(* IEC 61131-3 sources: json/test/Deserializer, 7 files *)

(* ---- Test_GetValues_Arrays.st ---- *)
USING Simatic.Ax.Conversion;
USING AxUnit.Assert;
USING System.Strings;
using Simatic.Ax.Json;

NAMESPACE Deserializer
NAMESPACE GetValues

{TestFixture}
CLASS Test_Deserializer_GetValues_Arrays
    VAR protected
        deserializer : Deserializer;

        buffer : ARRAY[0..999] OF CHAR;
        key: STRING;
        value: STRING;
    END_VAR

    {Test}
    Method Public Test_FindValue_in_JSON_SimpleArray
        VAR
            JSON_Entry: STRING := '{ "arraykey": [123, 456]}';

            len:DINT;
            keyFound: BOOL;
        END_VAR

        len:= Strings.ToArray(str := JSON_Entry, arr := buffer);
        deserializer.SetBuffer(REF(buffer)); //TODO: ausbauen und ersetzen durch buffer in methode

        key := 'arraykey';
        keyFound := deserializer.GetValue( REF(key), value);
        Equal('[123, 456]', value);
    END_Method

    {Test}
    Method Public Test_FindValue_in_JSON_ComplexArray
        VAR
            JSON_Entry: STRING := '{ "key1": 1234,"arraykey": [123, 456], "key2": 456}';

            len:DINT;
            keyFound: BOOL;
        END_VAR

        len:= Strings.ToArray(str := JSON_Entry, arr := buffer);
        deserializer.SetBuffer(REF(buffer)); //TODO: ausbauen und ersetzen durch buffer in methode

        key := 'arraykey';
        keyFound := deserializer.GetValue( REF(key), value);
        Equal('[123, 456]', value);
    END_Method

    {Test}
    Method Public Test_FindValue_in_JSON_NestedArray
        VAR
            JSON_Entry: STRING := '{ "key1": 1234,"arraykey": [{"nestedkey1": 1234, "nestedkey2": 456}, {"nestedkey3": 1234, "nestedkey4": 456}], "key2": 456}';

            len:DINT;
            keyFound: BOOL;
        END_VAR

        len:= Strings.ToArray(str := JSON_Entry, arr := buffer);
        deserializer.SetBuffer(REF(buffer)); //TODO: ausbauen und ersetzen durch buffer in methode

        key := 'arraykey';
        keyFound := deserializer.GetValue( REF(key), value);
        Equal('[{"nestedkey1": 1234, "nestedkey2": 456}, {"nestedkey3": 1234, "nestedkey4": 456}]', value);
    END_Method

END_CLASS

END_NAMESPACE
END_NAMESPACE

(* ---- Test_GetValues_NestedElements.st ---- *)
USING Simatic.Ax.Conversion;
USING AxUnit.Assert;
USING System.Strings;
using Simatic.Ax.Json;

NAMESPACE Deserializer
NAMESPACE GetValues

{TestFixture}
CLASS Test_Deserializer_GetValues_NestedElements
    VAR protected
        deserializer : Deserializer;

        buffer : ARRAY[0..999] OF CHAR;
        key: STRING;
        value: STRING;
    END_VAR

    {Test}
    Method Public Test_FindValue_in_JSON_NestedArray
        VAR
            JSON_Entry: STRING := '{ "key1": 1234,"arraykey": [{"nestedkey1": 1234, "nestedkey2": 456}, {"nestedkey3": 1234, "nestedkey4": 456}], "key2": 456}';

            len:DINT;
            keyFound: BOOL;
        END_VAR

        len:= Strings.ToArray(str := JSON_Entry, arr := buffer);
        deserializer.SetBuffer(REF(buffer)); //TODO: ausbauen und ersetzen durch buffer in methode

        key := 'arraykey';
        keyFound := deserializer.GetValue( REF(key), value);
        Equal('[{"nestedkey1": 1234, "nestedkey2": 456}, {"nestedkey3": 1234, "nestedkey4": 456}]', value);
    END_Method

    {Test}
    Method Public Test_FindValue_NestedElement_in_JSON_SimpleEntries
        VAR
            JSON_Entry: STRING := '{"key": {"nested1" : "hello", "nested2" : 1234  } }';
            len:DINT;
            keyFound: BOOL;
            nestedElement: STRING;
        END_VAR

        len:= Strings.ToArray(str := JSON_Entry, arr := buffer);
        deserializer.SetBuffer(REF(buffer));

        key := 'key';
        keyFound := deserializer.GetValue( REF(key), nestedElement);
        Equal(true, keyFound);
        Equal('{"nested1" : "hello", "nested2" : 1234  }', nestedElement);

        len := Strings.ToArray(str := nestedElement, arr := buffer);
        //deserializer.SetBuffer(REF(buffer));
        key := 'nested1';
        keyFound := deserializer.GetValue( REF(key), value);
        Equal('hello', value);

    END_Method

    {Test}
    Method Public Test_FindValue_NestedElement_in_JSON_MoreEntries
        VAR
            JSON_Entry: STRING := '{"anotherkey": 123, "key": {"nested1" : "hello", "nested2" : 1234  }, "differentKey": 12 }';
            len:DINT;
            keyFound: BOOL;
            nestedElement: STRING;
        END_VAR

        len:= Strings.ToArray(str := JSON_Entry, arr := buffer);
        deserializer.SetBuffer(REF(buffer));

        key := 'key';
        keyFound := deserializer.GetValue( REF(key), nestedElement);
        Equal(true, keyFound);
        Equal('{"nested1" : "hello", "nested2" : 1234  }', nestedElement);

        len := Strings.ToArray(str := nestedElement, arr := buffer);
        //deserializer.SetBuffer(REF(buffer));
        key := 'nested1';
        keyFound := deserializer.GetValue( REF(key), value);
        Equal('hello', value);

    END_Method

    {Test}
    Method Public Test_FindValue_NestedElement_in_JSON_ArrayInNested
        VAR
            JSON_Entry: STRING := '{"anotherkey": 123, "key": {"nested1" : ["hello", "123"], "nested2" : 1234  }, "differentKey": 12 }';
            len:DINT;
            keyFound: BOOL;
            nestedElement: STRING;
        END_VAR

        len:= Strings.ToArray(str := JSON_Entry, arr := buffer);
        deserializer.SetBuffer(REF(buffer));

        key := 'key';
        keyFound := deserializer.GetValue( REF(key), nestedElement);
        Equal(true, keyFound);
        Equal('{"nested1" : ["hello", "123"], "nested2" : 1234  }', nestedElement);

        len := Strings.ToArray(str := nestedElement, arr := buffer);
        //deserializer.SetBuffer(REF(buffer));
        key := 'nested1';
        keyFound := deserializer.GetValue( REF(key), value);
        Equal('["hello", "123"]', value);

    END_Method

END_CLASS

END_NAMESPACE
END_NAMESPACE

(* ---- Test_GetValuesFromIndex.st ---- *)
USING Simatic.Ax.Conversion;
USING AxUnit.Assert;
USING System.Strings;
using Simatic.Ax.Json;

NAMESPACE Deserializer
NAMESPACE GetValuesFromIndex

{TestFixture}
CLASS Test_Deserializer_GetValuesFromIndex
    VAR protected
        deserializer : Deserializer;

        buffer : ARRAY[0..999] OF CHAR;
        key: STRING;
        value: STRING;
        testIndex1: INT;
        testIndex2: INT;
    END_VAR

    {Test}
    Method Public Test_GetValueFromIndex_GetValue
        VAR
            len: DINT;
        END_VAR

        len:= Strings.ToArray(str := '1234', arr := buffer);
        deserializer.SetBuffer(REF(buffer));

        testIndex1:= 0; testIndex2 := 3;
        value:= deserializer.GetValueFromIndex(testIndex1, testIndex2);

        Equal('1234', value);

    END_Method

    {Test}
    Method Public Test_GetValueFromIndex_GetValue_withSpaces
        VAR
            len: DINT;
        END_VAR

        len:= Strings.ToArray(str := '    1234    ', arr := buffer);
        deserializer.SetBuffer(REF(buffer));

        testIndex1:= 0; testIndex2 := 10;
        value:= deserializer.GetValueFromIndex(testIndex1, testIndex2);

        Equal('1234', value);

    END_Method

    {Test}
    Method Public Test_GetValueFromIndex_GetValue_withQuotationMarks
        VAR
            len: DINT;
        END_VAR

        len:= Strings.ToArray(str := ' "1234"      ', arr := buffer);
        deserializer.SetBuffer(REF(buffer));

        testIndex1:= 0; testIndex2 := 10;
        value:= deserializer.GetValueFromIndex(testIndex1, testIndex2);

        Equal('1234', value);

    END_Method

END_CLASS

END_NAMESPACE
END_NAMESPACE

(* ---- Test_Playground.st ---- *)
USING Simatic.Ax.Conversion;
USING AxUnit.Assert;
USING System.Strings;
using Simatic.Ax.Json;

NAMESPACE Deserializer

{TestFixture}
CLASS Playground
    VAR protected
        deserializer : Deserializer;
        keyArray: ARRAY [0..1] OF STRING := ['key1', 'nestedkey1'];
        buffer : ARRAY[0..999] OF CHAR;
        value: STRING;
    END_VAR

    {Test}
    Method Public Test_FindValue_in_nestedElementWithPlayground
        VAR
            JSON_Entry: STRING := '{ "key1": {"nestedkey1": 123}}';
            len:DINT;
            keyFound: BOOL;
        END_VAR

        len:= Strings.ToArray(str := JSON_Entry, arr := buffer);
        deserializer.SetBuffer(REF(buffer)); //TODO: ausbauen und ersetzen durch buffer in methode

        keyFound := deserializer.GetValue_WithKeyArray( REF(keyArray), value);
        Equal('123', value);

    END_Method

END_CLASS

END_NAMESPACE

(* ---- Test_TryParse.st ---- *)
USING Simatic.Ax.Conversion;
USING AxUnit.Assert;
USING System.Strings;
using Simatic.Ax.Json;

NAMESPACE Deserializer

{TestFixture}
CLASS TryParse
    VAR protected
        deserializer : Deserializer;
        buffer : ARRAY[0..999] OF CHAR;
        value: STRING;
    END_VAR

    {Test}
    Method Public Test_TryParse_String
        VAR
            JSON_Entry: STRING := '{ "key1": {"nestedkey1": 123}}';
            key: STRING := 'key1';
            len:DINT;
            keyFound: BOOL;
        END_VAR

        len:= Strings.ToArray(str := JSON_Entry, arr := buffer);
        deserializer.SetBuffer(REF(buffer)); //TODO: ausbauen und ersetzen durch buffer in methode

        keyFound := deserializer.TryParse_STRING( key, value);
        Equal('{"nestedkey1": 123}', value);

    END_Method

    {Test}
    Method Public Test_TryParse_String_Nested
        VAR
            JSON_Entry: STRING := '{ "aKey": "hallo", "anotherKey": 1234, "key1": {"nestedkey1": 123, "nestedkey2": "hallo", "nestedkey3": {"nestedInNestedkey1": 1234 }}}';
            keyArray: ARRAY [0..1] OF STRING := ['key1', 'nestedkey1'];
            len:DINT;
            keyFound: BOOL;
        END_VAR

        len:= Strings.ToArray(str := JSON_Entry, arr := buffer);
        deserializer.SetBuffer(REF(buffer)); //TODO: ausbauen und ersetzen durch buffer in methode

        keyFound := deserializer.TryParse_STRING( keyArray, value);
        Equal('123', value);

    END_Method

END_CLASS

END_NAMESPACE

(* ---- TestFindCharacterInArray.st ---- *)
USING AxUnit.Assert;

NAMESPACE Simatic.Ax.Json

    {TestFixture}
    CLASS TestFindCharacterInArray
        VAR
            o : FindCharacterInArray;
            inputBuffer : ARRAY[0..99] OF CHAR;
            index : DINT;
            done, error : BOOL;
            cmd : IPlcOpen;
        END_VAR

        {Test (ExpectedIndex := 0)}
        {Test (ExpectedIndex := 1)}
        {Test (ExpectedIndex := 10)}
        {Test (ExpectedIndex := 99)}
        METHOD PUBLIC Find_start_Char_At_First_Position_Search_Forward
            VAR_INPUT
                ExpectedIndex : DINT;
            END_VAR
            inputBuffer[ExpectedIndex] := '{';
            cmd := o.Find(buffer := REF(inputBuffer), c := '{', mode := FindeMode#MODE_FORWARD);
            IF NOT cmd.Busy() THEN
                IF cmd.Done() THEN
                    index := o.GetIndex();
                    ; // command successfully done
                ELSIF cmd.Error() THEN
                    ; // error occured
                ELSIF cmd.Aborted() THEN
                    ; // command was aborted
                END_IF;
            ELSE
                ; // wait until it is not busy any more
            END_IF;
            Equal(expected := ExpectedIndex, actual := index);
            Equal(expected := FALSE, actual := error);
            Equal(expected := FALSE, actual := cmd.Error());
            done := cmd.Done();
            Equal(expected := TRUE, actual := done);
            Equal(expected := TRUE, actual := cmd.Done());
        END_METHOD

        {Test (ExpectedIndex := 0)}
        {Test (ExpectedIndex := 1)}
        {Test (ExpectedIndex := 10)}
        {Test (ExpectedIndex := 99)}
        METHOD PUBLIC Find_start_Char_At_First_Position_Search_Reverse
            VAR_INPUT
                ExpectedIndex : DINT;
            END_VAR
            inputBuffer[ExpectedIndex] := '{';
            cmd := o.Find(buffer := REF(inputBuffer), c := '{', mode := FindeMode#MODE_REVERSE);
            IF NOT cmd.Busy() THEN
                IF cmd.Done() THEN
                    index := o.GetIndex();
                    done := TRUE;
                    ; // command successfully done
                ELSIF cmd.Error() THEN
                    ; // error occured
                ELSIF cmd.Aborted() THEN
                    ; // command was aborted
                END_IF;
            ELSE
                ; // wait until it is not busy any more
            END_IF;
            Equal(expected := ExpectedIndex, actual := index);
            Equal(expected := FALSE, actual := error);
            Equal(expected := FALSE, actual := cmd.Error());
            Equal(expected := TRUE, actual := done);
            Equal(expected := TRUE, actual := cmd.Done());
        END_METHOD

        {Test}
        METHOD PUBLIC Error_Character_Not_Found
            cmd := o.Find(buffer := REF(inputBuffer), c := '{', mode := FindeMode#MODE_FORWARD);
            IF NOT cmd.Busy() THEN
                IF cmd.Done() THEN
                    index := o.GetIndex();
                    done := TRUE;
                    ; // command successfully done
                ELSIF cmd.Error() THEN
                    error := TRUE;
                    ; // error occured
                END_IF;
            ELSE
                ; // wait until it is not busy any more
            END_IF;
            Equal(expected := 0, actual := index);
            Equal(expected := TRUE, actual := error);
            Equal(expected := TRUE, actual := cmd.Error());
            Equal(expected := FALSE, actual := cmd.Done());
            ;
        END_METHOD
    END_CLASS

END_NAMESPACE

(* ---- TestFindKeyInBuffer.st ---- *)
USING Simatic.Ax.Conversion;
USING AxUnit.Assert;
USING System.Strings;
using Simatic.Ax.Json;

NAMESPACE Deserializer
NAMESPACE FindKeys

{TestFixture}
CLASS Test_FindKeyInBuffer
    VAR protected
        deserializer : Deserializer;

        buffer : ARRAY[0..999] OF CHAR;
        key: STRING;
        value: STRING;
        testIndex1: INT;
        testIndex2: INT;
    END_VAR

    {Test}
    Method Public Test_FindKeysPosition_in_JSON_SimpleEntries
        VAR
            JSON_Entry: STRING := '{"key ": " Elem ent1", "Hello": "something", "Nothing": 456, "Key 2": 1234 }';

            len:DINT;
            keyStart : int;
            keyEnd : int;
            keyFound: BOOL;
        END_VAR

        len:= Strings.ToArray(str := JSON_Entry, arr := buffer);
        deserializer.SetBuffer(REF(buffer));

        key := 'key ';
        keyFound := deserializer.TryParse( key, value);
        Equal(TRUE, keyFound);

        key := 'Key 2';
        keyFound := deserializer.TryParse( key, value);
        Equal(TRUE, keyFound);

        key := 'not a key';
        keyFound := deserializer.TryParse( key, value);
        Equal(FALSE, keyFound);
    END_Method

    {Test}
    Method Public Test_FindKeysPosition_in_JSON_Single_Nested_Entry
        VAR
            JSON_Entry: STRING := '{"nested": {"nested1" : "hello", "nested2" : 1234  }}';

            len:DINT;
            keyStart : int;
            keyEnd : int;
            keyFound: BOOL;
        END_VAR

        len:= Strings.ToArray(str := JSON_Entry, arr := buffer);
        deserializer.SetBuffer(REF(buffer));

        key := 'nested';
        keyFound := deserializer.TryParse( key, value);
        Equal(TRUE, keyFound);
    END_Method

    {Test}
    Method Public Test_FindKeysPosition_with_JSON_Nested_Entry
        VAR
            JSON_Entry: STRING := '{"key ": " Elem ent1", "nested": {"nested1" : "hello", "nested2" : 1234  }, "key2": " Elem ent1"}';

            len:DINT;
            keyStart : int;
            keyEnd : int;
            keyFound: BOOL;
        END_VAR

        len:= Strings.ToArray(str := JSON_Entry, arr := buffer);
        deserializer.SetBuffer(REF(buffer));

        key := 'key ';
        keyFound := deserializer.TryParse( key, value);
        Equal(TRUE, keyFound);

        key := 'nested';
        keyFound := deserializer.TryParse( key, value);
        Equal(TRUE, keyFound);

        key := 'key2';
        keyFound := deserializer.TryParse( key, value);
        Equal(TRUE, keyFound);
    END_Method

    {Test}
    Method Public Test_FindKeysPosition_with_JSON_SimpleArray
        VAR
            JSON_Entry: STRING := '{ "simpleArray": [123, 456]}';

            len:DINT;
            keyStart : int;
            keyEnd : int;
            keyFound: BOOL;
        END_VAR

        len:= Strings.ToArray(str := JSON_Entry, arr := buffer);
        deserializer.SetBuffer(REF(buffer));

        key := 'simpleArray';
        keyFound := deserializer.TryParse( key, value);
        Equal(TRUE, keyFound);
    END_Method

    {Test}
    Method Public Test_KeyIsInIndexSpan_FindsKey
        VAR
            len:DINT;
            keyStart : int := 0;
            keyEnd : int := 2;
            keyFound: BOOL;
        END_VAR

        key := 'key';
        len:= Strings.ToArray(str := key, arr := buffer);
        deserializer.SetBuffer(REF(buffer));

        keyFound := deserializer.KeyIsInIndexSpan(key, keyStart, keyEnd);
        Equal(TRUE, keyFound);

        key := 'not';
        keyFound := deserializer.KeyIsInIndexSpan(key, keyStart, keyEnd);
        Equal(FALSE, keyFound);
    END_Method

END_CLASS

END_NAMESPACE
END_NAMESPACE
